TYPE ToolStorage :
STRUCT
	eoatA_pos1 : BOOL;
	eoatB_pos1 : BOOL;
	
	eoatA_pos2 : BOOL;
	eoatB_pos2 : BOOL;	
END_STRUCT
END_TYPE

(* stored: Version 1.1.0.1, ProductVersion 3.1.4024.11
   DUT ToolStorage: Id {2dc4acc1-5d39-4b0a-8c99-9c231c4d3c98} *)
